{attribute 'linkalways'} 
{attribute 'no_explicit_call' := 'This FB is a CLASS and must be accessed using methods or properties'}
{attribute 'enable_dynamic_creation'}
FUNCTION_BLOCK _Array0to1OfREAL EXTENDS ArrayDatatypeBase_1D
VAR CONSTANT
	lBound : DINT := 0;
	uBound : DINT := 1;
END_VAR
VAR
	localData : ARRAY [lBound..uBound] OF REAL;
	activeData : REFERENCE TO ARRAY [lBound..uBound] OF REAL REF= localData;
	elements : ARRAY [lBound..uBound] OF _REAL(0.0);
	baseType : _REAL(0.0);
END_VAR

PROPERTY PUBLIC Address : PVOID
GET
Address := ADR(activeData);
END_GET
END_PROPERTY

PROPERTY PUBLIC BaseDatatype : I_Datatype
GET
BaseDatatype := baseType;
END_GET
END_PROPERTY

METHOD PUBLIC ClearReference
VAR_INPUT
END_VAR
activeData REF= localData;
SetElementReference();
END_METHOD

METHOD PUBLIC Clone : I_Datatype
VAR
    pClone : POINTER TO _Array0to1OfREAL;
END_VAR
pClone := __NEW(_Array0to1OfREAL());
pClone^.Value := Value;
Clone := pClone^;
END_METHOD

METHOD FB_init : BOOL
VAR_INPUT
	bInitRetains : BOOL; // if TRUE, the retain variables are initialized (warm start / cold start)
	bInCopyCode : BOOL;  // if TRUE, the instance afterwards gets moved into the copy code (online change)
END_VAR
SetElementReference();
END_METHOD

METHOD PUBLIC MakeReferenceTo
VAR_INPUT
	ReferenceTarget : REFERENCE TO ARRAY [lBound..uBound] OF REAL;
END_VAR
activeData REF= ReferenceTarget;
SetElementReference();
END_METHOD

METHOD PROTECTED OnSerializeArrayValues
VAR_INPUT
	Serializer : I_Serializer;
END_VAR
VAR
	i : DINT;
END_VAR
FOR i := lBound TO uBound DO
	elements[i].SerializeWith(Serializer);
END_FOR
END_METHOD

METHOD PROTECTED SetElementReference
VAR_INPUT
END_VAR
VAR
	i : DINT;
END_VAR
FOR i := lBound TO uBound DO
	elements[i].MakeReferenceTo(activeData[i]);
END_FOR
END_METHOD

PROPERTY PUBLIC Size : UDINT
GET
Size := SIZEOF(activeData);
END_GET
END_PROPERTY

METHOD PROTECTED TryDeserializeArrayValues : BOOL
VAR_INPUT
	Deserializer : I_Deserializer;
	Feedback : I_DeserializerFeedback;
END_VAR
VAR
	enumerator : I_DeserializerArrayForwardEnumerator;
	i : DINT;
END_VAR
enumerator := Deserializer.GetArrayEnumerator();
i := lBound;

WHILE enumerator.MoveNext() AND i <= uBound DO
	
	IF NOT elements[i].TryDeserializeFrom(enumerator.Current, Feedback) THEN
		EXIT;
	END_IF
	i := i + 1;

END_WHILE
enumerator.Dispose();
END_METHOD

METHOD PUBLIC TryGetElementAsDatatypeByIndex : BOOL
VAR_INPUT
	Index : DINT;
	Destination : REFERENCE TO I_Datatype;
END_VAR
IF Index < lbound OR Index > ubound THEN
	RETURN;
END_IF

Destination := elements[Index];
TryGetElementAsDatatypeByIndex := TRUE;
END_METHOD

METHOD PUBLIC TryGetLowerBound : BOOL
VAR_INPUT
	Dimention : UDINT;
	Destination : REFERENCE TO DINT;
END_VAR
IF Dimention = 1 THEN
	Destination := lBound;
	TryGetLowerBound := TRUE;
END_IF
END_METHOD

METHOD PUBLIC TryGetUpperBound : BOOL
VAR_INPUT
	Dimention : UDINT;
	Destination : REFERENCE TO DINT;
END_VAR
IF Dimention = 1 THEN
	Destination := uBound;
	TryGetUpperBound := TRUE;
END_IF
END_METHOD

METHOD TryMakeReferenceTo : BOOL
VAR_INPUT
	Target : I_Datatype;
END_VAR
VAR
	targetAsArray : I_ArrayDatatype;
	pTargetData : POINTER TO ARRAY [lBound..uBound] OF REAL;
END_VAR
IF NOT Target.TryResolveAsArrayDatatype(targetAsArray) THEN
	RETURN;
END_IF

IF NOT (targetAsArray.Identifier = Identifier) THEN
	RETURN;
END_IF

pTargetData := Target.Address;
activeData REF= pTargetData^;
SetElementReference();
TryMakeReferenceTo := TRUE;
END_METHOD

PROPERTY PUBLIC Value : REFERENCE TO ARRAY [lBound..uBound] OF REAL;
GET
Value ref= activeData;
END_GET
END_PROPERTY

END_FUNCTION_BLOCK

(* stored: Version 1.1.0.1, ProductVersion 3.1.4024.13
   POU _Array0to1OfREAL: Id {d3dadfee-0c1a-03df-127d-b2f699ba5ef6}, SpecialFunc None
   Folder Core: Id {5d997022-646e-0aa3-26ff-7f22363942ea}
   Folder Constructor: Id {227057ae-2a92-0cc6-203d-fd4e94edbb08}
   Folder Protected: Id {02c5c413-4af4-0ef0-32f1-9a3c9c8cb581}
   Folder Customize: Id {51d6a80b-fcf9-0ae8-10a9-d4a52264ed7e}
   Property Address: Id {b70eb4fe-6e84-0448-06ab-7587bdbb2bec}
   Get Get: Id {0011f921-2200-054b-3436-15966d7c36ea}
   Property BaseDatatype: Id {8bfcf251-8fef-0cbe-3412-4ea85ee46b63}
   Get Get: Id {0a467fd2-9db5-0c54-0c44-b08162b0e311}
   Method ClearReference: Id {5fe1586f-c9c0-0f29-27c6-8dcef33452d7}
   Method Clone: Id {24148a2f-a3a5-0994-3e19-a4553ab4df24}
   Method FB_init: Id {6f0ae0e1-627a-053a-0cc1-01c4b7c02bdc}
   Method MakeReferenceTo: Id {64d32564-a6ec-082f-026b-956cc935b508}
   Method OnSerializeArrayValues: Id {0583b999-b15f-0d42-0222-b85febcc7fd5}
   Method SetElementReference: Id {588fdd22-3bcb-06d3-17a3-bd51260213c4}
   Property Size: Id {a03c556b-4f1c-0a46-1e49-ae73e90780c7}
   Get Get: Id {56da5978-1bd1-09de-00ae-79672bb417c9}
   Method TryDeserializeArrayValues: Id {3c7117ea-37bd-0382-2de2-e4b6dbd98ff5}
   Method TryGetElementAsDatatypeByIndex: Id {174a7c61-a37f-0de4-130d-10837880aa4c}
   Method TryGetLowerBound: Id {545a83f6-e416-0006-11ec-ba6722146d6d}
   Method TryGetUpperBound: Id {9de01636-ceae-01d0-2c0e-6572de383812}
   Method TryMakeReferenceTo: Id {58d26488-71e9-0ea2-1015-11e40f2593e9}
   Property Value: Id {efd120f4-ca55-00bc-2618-fe8a4436221b}
   Get Get: Id {1f4c9c75-1e4e-0ae4-102a-b45cb62c6fb0} *)
